(* CoDeSys 2.3.9.41 project: Basics_Test.pro *)
(* Libraries: STANDARD.LIB 5.6.98 11:03:02 *)

(* Task configuration *)
TASK MY_TASK (PRIORITY := 0, INTERVAL := T#1ms);
	MAIN
END_TASK

(* Global variable list: Global_Variables *)
VAR_GLOBAL
	rV3 : REAL := -1.5;
END_VAR

(* POU MAIN, ST *)
PROGRAM MAIN
VAR
	rV1 : REAL := 3.1;
	rV2 : REAL := 7.7;
	mep : MEINE_MEP_FUNKTION_1;
END_VAR
mep(rPAR1 := rV1, rPAR2 := rV2);
rV3 := mep.rOUT;
END_PROGRAM

(* POU MEINE_MEP_FUNKTION_1, ST *)
FUNCTION_BLOCK MEINE_MEP_FUNKTION_1
VAR_INPUT
	rPAR1 : REAL;
	rPAR2 : REAL;
END_VAR
VAR_OUTPUT
	rOUT : REAL;
END_VAR
VAR
END_VAR
rOUT := rPAR1 + rPAR2 + rOUT;
END_FUNCTION_BLOCK
